{attribute 'GeneratedUsingTerminal: ELX9560-0000-0018'}
{attribute addProperty BoxType "ELX9560-0000-0018"}
{attribute addProperty Id "Uin_OKAT %I*BOOL1"}
{attribute addProperty CRC "1652344174"}
{attribute addProperty Size "1"}
TYPE Status_Uin_627CC56E :
STRUCT
	{attribute addProperty Name "Uin_OK"}
	Uin_OK AT %I* : BOOL;
END_STRUCT
END_TYPE

(* stored: Version 1.2.0.0, ProductVersion 3.1.4024.9
   DUT Status_Uin_627CC56E: Id {4d572e8b-eea1-4fcd-b095-863aeacac746} *)
